(* IEC 61131-3 sources: CodesysTest/alpha/export/FBs/Unused/ElectricPressureBarFB.pou, 2 files *)

(* ---- AutoOpenJaw.m.st ---- *)
(*#-#-#-#-#-#-#-#-#-#---Declaration---#-#-#-#-#-#-#-#-#-#-#-#-#*)

METHOD AutoOpenJaw
VAR_INPUT
END_VAR
(*#-#-#-#-#-#-#-#-#-#---Implementation---#-#-#-#-#-#-#-#-#-#-#-#-#*)

_amOpenJaw := TRUE;

(* ---- ClearCommands.m.st ---- *)
(*#-#-#-#-#-#-#-#-#-#---Declaration---#-#-#-#-#-#-#-#-#-#-#-#-#*)

METHOD PRIVATE ClearCommands
VAR_INPUT
END_VAR
(*#-#-#-#-#-#-#-#-#-#---Implementation---#-#-#-#-#-#-#-#-#-#-#-#-#*)

_amCloseJaw := FALSE;
_amOpenJaw := FALSE;
